// TIA Portal V20 export
TYPE "LER_typeVisionGapResultData"
// stored: Access Published
   STRUCT
      visionLengthOfSeparatorCathodeJudgementResult : Real;   // Vision Length of Separator Cathode Judgement Result (0:NONE,1:OK,2:NG)
      visionLengthOfSeparatorAnodeJudgementResult : Real;   // Vision Length of Separator Anode Judgement Result (0:NONE,1:OK,2:NG)
      visionCathodeLengthJudgementResult : Real;   // Vision Cathode Length Judgement Result (0:NONE,1:OK,2:NG)
      visionAnodeLengthJudgementResult : Real;   // Vision Anode Length Judgement Result (0:NONE,1:OK,2:NG)
      visionCathodeToSeparatorY1JudgementResult : Real;   // Vision Cathode to Separator Y1 Judgement Result (0:NONE,1:OK,2:NG)
      visionCathodeToSeparatorY2JudgementResult : Real;   // Vision Cathode to Separator Y2 Judgement Result (0:NONE,1:OK,2:NG)
      visionCathodeToSeparatorY3JudgementResult : Real;   // Vision Cathode to Separator Y3 Judgement Result (0:NONE,1:OK,2:NG)
      visionCathodeToSeparatorY4JudgementResult : Real;   // Vision Cathode to Separator Y4 Judgement Result (0:NONE,1:OK,2:NG)
      visionCathodeToAnodeY1JudgementResult : Real;   // Vision Cathode to Anode Y1 Judgement Result (0:NONE,1:OK,2:NG)
      visionCathodeToAnodeY2JudgementResult : Real;   // Vision Cathode to Anode Y2 Judgement Result (0:NONE,1:OK,2:NG)
      visionAnodeToCathodeY1JudgementResult : Real;   // Vision Anode to Cathode Y1 Judgement Result (0:NONE,1:OK,2:NG)
      visionAnodeToCathodeY2JudgementResult : Real;   // Vision Anode to Cathode Y2 Judgement Result (0:NONE,1:OK,2:NG)
      visionAnodeToSeparatorY1JudgementResult : Real;   // Vision Anode to Separator Y1 Judgement Result (0:NONE,1:OK,2:NG)
      visionAnodeToSeparatorY2JudgementResult : Real;   // Vision Anode to Separator Y2 Judgement Result (0:NONE,1:OK,2:NG)
      visionAnodeToCathodeX1JudgementResult : Real;   // Vision Anode to Cathode X1 Judgement Result (0:NONE,1:OK,2:NG)
      visionAnodeToCathodeX2JudgementResult : Real;   // Vision Anode to Cathode X2 Judgement Result (0:NONE,1:OK,2:NG)
      visionAnodeToCathodeX3JudgementResult : Real;   // Vision Anode to Cathode X3 Judgement Result (0:NONE,1:OK,2:NG)
      visionAnodeToCathodeX4JudgementResult : Real;   // Vision Anode to Cathode X4 Judgement Result (0:NONE,1:OK,2:NG)
      visionCathodeToSeparatorX1JudgementResult : Real;   // Vision Cathode to Separator X1 Judgement Result (0:NONE,1:OK,2:NG)
      visionCathodeToSeparatorX2JudgementResult : Real;   // Vision Cathode to Separator X2 Judgement Result (0:NONE,1:OK,2:NG)
      visionCathodeToSeparatorX3JudgementResult : Real;   // Vision Cathode to Separator X3 Judgement Result (0:NONE,1:OK,2:NG)
      visionCathodeToSeparatorX4JudgementResult : Real;   // Vision Cathode to Separator X4 Judgement Result (0:NONE,1:OK,2:NG)
      visionAnodeToSeparatorX1JudgementResult : Real;   // Vision Anode to Separator X1 Judgement Result (0:NONE,1:OK,2:NG)
      visionAnodeToSeparatorX2JudgementResult : Real;   // Vision Anode to Separator X2 Judgement Result (0:NONE,1:OK,2:NG)
      visionAnodeToSeparatorX3JudgementResult : Real;   // Vision Anode to Separator X3 Judgement Result (0:NONE,1:OK,2:NG)
      visionAnodeToSeparatorX4JudgementResult : Real;   // Vision Anode to Separator X4 Judgement Result (0:NONE,1:OK,2:NG)
      visionLengthOfSeparatorCathodeReply : Real;   // Vision Length of Separator Cathode_Reply [mm](1/1000)
      visionLengthOfSeparatorCathodeUpperRangeReply : Real;   // Vision Length of Separator Cathode Upper Range Reply [mm](1/1000)
      visionLengthOfSeparatorCathodeLowerRangeReply : Real;   // Vision Length of Separator Cathode Lower Range Reply [mm](1/1000)
      visionLengthOfSeparatorAnodeReply : Real;   // Vision Length of Separator Anode Reply [mm](1/1000)
      visionLengthOfSeparatorAnodeUpperRangeReply : Real;   // Vision Length of Separator Anode Upper Range Reply [mm](1/1000)
      visionLengthOfSeparatorAnodeLowerRangeReply : Real;   // Vision Length of Separator Anode Lower Range Reply [mm](1/1000)
      visionCathodeLengthReply : Real;   // Vision Cathode Length Reply [mm](1/1000)
      visionCathodeLengthUpperRangeReply : Real;   // Vision Cathode Length(1/1000) Upper Range Reply [mm](1/1000)
      visionCathodeLengthLowerRangeReply : Real;   // Vision Cathode Length(1/1000) Lower Range Reply [mm](1/1000)
      visionAnodeLengthReply : Real;   // Vision Anode Length Reply [mm](1/1000)
      visionAnodeLengthUpperRangeReply : Real;   // Vision Anode Length(1/1000) Upper Range Reply [mm](1/1000)
      visionAnodeLengthLowerRangeReply : Real;   // Vision Anode Length(1/1000) Lower Range Reply [mm](1/1000)
      visionCathodeToSeparatorY1Reply : Real;   // Vision Cathode to Separator Y1 Reply [mm](1/1000)
      visionCathodeToSeparatorY1UpperRangeReply : Real;   // Vision Cathode to Separator Y1(1/1000) Upper Range Reply [mm](1/1000)
      visionCathodeToSeparatorY1LowerRangeReply : Real;   // Vision Cathode to Separator Y1(1/1000) Lower Range Reply [mm](1/1000)
      visionCathodeToSeparatorY2Reply : Real;   // Vision Cathode to Separator Y2 Reply [mm](1/1000)
      visionCathodeToSeparatorY2UpperRangeReply : Real;   // Vision Cathode to Separator Y2(1/1000) Upper Range Reply [mm](1/1000)
      visionCathodeToSeparatorY2LowerRangeReply : Real;   // Vision Cathode to Separator Y2(1/1000) Lower Range Reply [mm](1/1000)
      visionCathodeToSeparatorY3Reply : Real;   // Vision Cathode to Separator Y3 Reply [mm](1/1000)
      visionCathodeToSeparatorY3UpperRangeReply : Real;   // Vision Cathode to Separator Y3(1/1000) Upper Range Reply [mm](1/1000)
      visionCathodeToSeparatorY3LowerRangeReply : Real;   // Vision Cathode to Separator Y3(1/1000) Lower Range Reply [mm](1/1000)
      visionCathodeToSeparatorY4Reply : Real;   // Vision Cathode to Separator Y4 Reply [mm](1/1000)
      visionCathodeToSeparatorY4UpperRangeReply : Real;   // Vision Cathode to Separator Y4(1/1000) Upper Range Reply [mm](1/1000)
      visionCathodeToSeparatorY4LowerRangeReply : Real;   // Vision Cathode to Separator Y4(1/1000) Lower Range Reply [mm](1/1000)
      visionCathodeToAnodeY1Reply : Real;   // Vision Cathode to Anode Y1 Reply [mm](1/1000)
      visionCathodeToAnodeY1UpperRangeReply : Real;   // Vision Cathode to Anode Y1(1/1000) Upper Range Reply [mm](1/1000)
      visionCathodeToAnodeY1LowerRangeReply : Real;   // Vision Cathode to Anode Y1(1/1000) Lower Range Reply [mm](1/1000)
      visionCathodeToAnodeY2Reply : Real;   // Vision Cathode to Anode Y2 Reply [mm](1/1000)
      visionCathodeToAnodeY2UpperRangeReply : Real;   // Vision Cathode to Anode Y2(1/1000) Upper Range Reply [mm](1/1000)
      visionCathodeToAnodeY2LowerRangeReply : Real;   // Vision Cathode to Anode Y2(1/1000) Lower Range Reply [mm](1/1000)
      visionAnodeToCathodeY1Reply : Real;   // Vision Anode to Cathode Y1 Reply [mm](1/1000)
      visionAnodeToCathodeY1UpperRangeReply : Real;   // Vision Anode to Cathode Y1(1/1000) Upper Range Reply [mm](1/1000)
      visionAnodeToCathodeY1LowerRangeReply : Real;   // Vision Anode to Cathode Y1(1/1000) Lower Range Reply [mm](1/1000)
      visionAnodeToCathodeY2Reply : Real;   // Vision Anode to Cathode Y2 Reply [mm](1/1000)
      visionAnodeToCathodeY2UpperRangeReply : Real;   // Vision Anode to Cathode Y2(1/1000) Upper Range Reply [mm](1/1000)
      visionAnodeToCathodeY2LowerRangeReply : Real;   // Vision Anode to Cathode Y2(1/1000) Lower Range Reply [mm](1/1000)
      visionAnodeToSeparatorY1Reply : Real;   // Vision Anode to Separator Y1 Reply [mm](1/1000)
      visionAnodeToSeparatorY1UpperRangeReply : Real;   // Vision Anode to Separator Y1(1/1000) Upper Range Reply [mm](1/1000)
      visionAnodeToSeparatorY1LowerRangeReply : Real;   // Vision Anode to Separator Y1(1/1000) Lower Range Reply [mm](1/1000)
      visionAnodeToSeparatorY2Reply : Real;   // Vision Anode to Separator Y2 Reply [mm](1/1000)
      visionAnodeToSeparatorY2UpperRangeReply : Real;   // Vision Anode to Separator Y2(1/1000) Upper Range Reply [mm](1/1000)
      visionAnodeToSeparatorY2LowerRangeReply : Real;   // Vision Anode to Separator Y2(1/1000) Lower Range Reply [mm](1/1000)
      visionAnodeToCathodeX1Reply : Real;   // Vision Anode to Cathode X1 Reply [mm](1/1000)
      visionAnodeToCathodeX1UpperRangeReply : Real;   // Vision Anode to Cathode X1(1/1000) Upper Range Reply [mm](1/1000)
      visionAnodeToCathodeX1LowerRangeReply : Real;   // Vision Anode to Cathode X1(1/1000) Lower Range Reply [mm](1/1000)
      visionAnodeToCathodeX2Reply : Real;   // Vision Anode to Cathode X2 Reply [mm](1/1000)
      visionAnodeToCathodeX2UpperRangeReply : Real;   // Vision Anode to Cathode X2(1/1000) Upper Range Reply [mm](1/1000)
      visionAnodeToCathodeX2LowerRangeReply : Real;   // Vision Anode to Cathode X2(1/1000) Lower Range Reply [mm](1/1000)
      visionAnodeToCathodeX3Reply : Real;   // Vision Anode to Cathode X3 Reply [mm](1/1000)
      visionAnodeToCathodeX3UpperRangeReply : Real;   // Vision Anode to Cathode X3(1/1000) Upper Range Reply [mm](1/1000)
      visionAnodeToCathodeX3LowerRangeReply : Real;   // Vision Anode to Cathode X3(1/1000) Lower Range Reply [mm](1/1000)
      visionAnodeToCathodeX4Reply : Real;   // Vision Anode to Cathode X4 Reply [mm](1/1000)
      visionAnodeToCathodeX4UpperRangeReply : Real;   // Vision Anode to Cathode X4(1/1000) Upper Range Reply [mm](1/1000)
      visionAnodeToCathodeX4LowerRangeReply : Real;   // Vision Anode to Cathode X4(1/1000) Lower Range Reply [mm](1/1000)
      visionCathodeToSeparatorX1Reply : Real;   // Vision Cathode to Separator X1 Reply [mm](1/1000)
      visionCathodeToSeparatorX1UpperRangeReply : Real;   // Vision Cathode to Separator X1(1/1000) Upper Range Reply [mm](1/1000)
      visionCathodeToSeparatorX1LowerRangeReply : Real;   // Vision Cathode to Separator X1(1/1000) Lower Range Reply [mm](1/1000)
      visionCathodeToSeparatorX2Reply : Real;   // Vision Cathode to Separator X2 Reply [mm](1/1000)
      visionCathodeToSeparatorX2UpperRangeReply : Real;   // Vision Cathode to Separator X2(1/1000) Upper Range Reply [mm](1/1000)
      visionCathodeToSeparatorX2LowerRangeReply : Real;   // Vision Cathode to Separator X2(1/1000) Lower Range Reply [mm](1/1000)
      visionCathodeToSeparatorX3Reply : Real;   // Vision Cathode to Separator X3 Reply [mm](1/1000)
      visionCathodeToSeparatorX3UpperRangeReply : Real;   // Vision Cathode to Separator X3(1/1000) Upper Range Reply [mm](1/1000)
      visionCathodeToSeparatorX3LowerRangeReply : Real;   // Vision Cathode to Separator X3(1/1000) Lower Range Reply [mm](1/1000)
      visionCathodeToSeparatorX4Reply : Real;   // Vision Cathode to Separator X4 Reply [mm](1/1000)
      visionCathodeToSeparatorX4UpperRangeReply : Real;   // Vision Cathode to Separator X4(1/1000) Upper Range Reply [mm](1/1000)
      visionCathodeToSeparatorX4LowerRangeReply : Real;   // Vision Cathode to Separator X4(1/1000) Lower Range Reply [mm](1/1000)
      visionAnodeToSeparatorX1Reply : Real;   // Vision Anode to Separator X1 Reply [mm](1/1000)
      visionAnodeToSeparatorX1UpperRangeReply : Real;   // Vision Anode to Separator X1(1/1000) Upper Range Reply [mm](1/1000)
      visionAnodeToSeparatorX1LowerRangeReply : Real;   // Vision Anode to Separator X1(1/1000) Lower Range Reply [mm](1/1000)
      visionAnodeToSeparatorX2Reply : Real;   // Vision Anode to Separator X2 Reply [mm](1/1000)
      visionAnodeToSeparatorX2UpperRangeReply : Real;   // Vision Anode to Separator X2(1/1000) Upper Range Reply [mm](1/1000)
      visionAnodeToSeparatorX2LowerRangeReply : Real;   // Vision Anode to Separator X2(1/1000) Lower Range Reply [mm](1/1000)
      visionAnodeToSeparatorX3Reply : Real;   // Vision Anode to Separator X3 Reply [mm](1/1000)
      visionAnodeToSeparatorX3UpperRangeReply : Real;   // Vision Anode to Separator X3(1/1000) Upper Range Reply [mm](1/1000)
      visionAnodeToSeparatorX3LowerRangeReply : Real;   // Vision Anode to Separator X1(1/1000) Lower Range Reply [mm](1/1000)
      visionAnodeToSeparatorX4Reply : Real;   // Vision Anode to Separator X1 Reply [mm](1/1000)
      visionAnodeToSeparatorX4UpperRangeReply : Real;   // Vision Anode to Separator X1(1/1000) Upper Range Reply [mm](1/1000)
      visionAnodeToSeparatorX4LowerRangeReply : Real;   // Vision Anode to Separator X1(1/1000) Lower Range Reply [mm](1/1000)
   END_STRUCT;
END_TYPE
